INTERFACE I_Metadata EXTENDS I_Disposable, I_Serializable

METHOD PUBLIC Accept
VAR_INPUT
	Visitor : I_MetadataVisitor;
END_VAR
END_METHOD

PROPERTY PUBLIC Name : T_MAXSTRING
GET
END_GET
END_PROPERTY

METHOD PUBLIC SerializeWith
VAR_INPUT
	Serializer : I_Serializer;
END_VAR
END_METHOD

END_INTERFACE

(* stored: Version 1.1.0.1, ProductVersion 3.1.4024.12
   Itf I_Metadata: Id {df609e72-1d9f-06c6-38ef-3e2c502eecb5}
   Method Accept: Id {2f93461b-a249-003f-1afe-030a70299e97}
   Property Name: Id {bd30d1f5-cb2c-0a39-20d1-88b5a595317a}
   Get Get: Id {36ec1b28-5847-01dc-029f-8f90b43dbb11}
   Method SerializeWith: Id {adc764b8-5070-077e-06e5-40a6a5bee5ed} *)
